# EPICS autosave request: calcApp/Db/editSseq_settings.req
$(P)$(Q)Debug
$(P)$(Q)recordName
